{attribute addProperty BoxType "EP7402-0057-0017"}
{attribute addProperty Id "A_0055_EP7402_0057_0018EP7402_B02F38FD54468"}
{attribute addProperty CRC "1152328620"}
{attribute addProperty SizeInBites "544"}
{attribute addProperty SizeInBytes "68"}
TYPE A_0054_EP7402_0057_0017_44AF23AC EXTENDS EP7402_B02F38FD :
STRUCT
	{attribute addProperty Name "A_0055_EP7402_0057_0018"}
	A_0055_EP7402_0057_0018 : EP7402_B02F38FD;
END_STRUCT
END_TYPE

(* stored: Version 1.2.0.0, ProductVersion 3.1.4024.9
   DUT A_0054_EP7402_0057_0017_44AF23AC: Id {1a332261-2e9a-4d75-85c5-9e05b13ba549} *)
